GLOBALCONSTANTS DefaultPool_PWM (* Global constants *)
  PACKAGE Uebungen::const::UT;
  VAR_GLOBAL CONSTANT
    ISO_DESIGNATOR_WIDTH : UINT := 160;
    ISO_DESIGNATOR_HEIGHT : UINT := 80;
    ISO_MASK_SIZE : UINT := 480;
    ISO_VERSION_LABEL : STRING;
    MASK_WIDTH : UINT := 480;
    MASK_HEIGHT : UINT := 480;
    WorkingSet_0 : UINT := 0;
    Macro_100_perc : UINT := 1;
    Macro_050_perc : UINT := 2;
    Macro_075_perc : UINT := 3;
    Macro_000_perc : UINT := 4;
    Macro_025_perc : UINT := 5;
    DataMask_1000 : UINT := 1000;
    Button_050_perc : UINT := 6000;
    Button_075_perc : UINT := 6001;
    Button_000_perc : UINT := 6002;
    Button_025_perc : UINT := 6003;
    Button_100_perc : UINT := 6006;
    InputNumber_PWM_DUTY : UINT := 9000;
    InputNumber_PWM_Value : UINT := 9001;
    OutputString_percent : UINT := 11005;
    OutputString_WS : UINT := 11500;
    OutputNumber_100 : UINT := 12000;
    OutputNumber_8129 : UINT := 12001;
    OutputNumber_050 : UINT := 12002;
    OutputNumber_075 : UINT := 12003;
    OutputNumber_000 : UINT := 12004;
    OutputNumber_025 : UINT := 12005;
    Meter_17000 : UINT := 17000;
    LinearBargraph_18000 : UINT := 18000;
    ArchedBargraph_19000 : UINT := 19000;
    NumberVariable_PWM_Value : UINT := 21001;
    FontAttributes_12x16 : UINT := 23000;
    FontAttributes_12x16_B : UINT := 23001;
    FontAttributes_16x16 : UINT := 23004;
    FontAttributes_WS : UINT := 23500;
  END_VAR
END_GLOBALCONSTANTS
